(* Schneider Machine Expert - Basic project Ladder Programming_Devin Ezekiel Purba_2106701583, file version 2.7.0.0 *)
(* ProjectInformations: Name=New project *)

HARDWARE
  Cpu 0: TM221C16R
  EthernetConfiguration: NetworkName=M221, IpAllocationMode=FixedAddress, IpAddress=0.0.0.0, SubnetMask=0.0.0.0
  SerialLineConfiguration: Baud=Baud19200, Parity=ParityEven, DataBits=DataBits8, StopBits=StopBits1, PhysicalMedium=PhysicalMediumRs485, TransmissionMode=TransmissionModeModbusRtu, SlaveId=1, Addressing=SlaveAddressing
  MastTask: UsePeriodScanMode=false, PeriodScan=100
  FastTask: Period=255
  CpuBehavior: StartingMode=StartAsPreviousState, AutoSaveRamOnEeprom=true, WatchdogPeriod=250

SYMBOLS  (address, symbol, comment, settings)
  %M0       RUNNING
  %M1       MC_1_BUSY
  %M2       RETRO_1
  %M3       MC_2_BUSY
  %M4       RETRO_2
  %M5       MC_3_BUSY
  %M6       RETRO_5
  %M7       MC_4_BUSY
  %M8       RETRO_6
  %M9       MC_5_BUSY
  %M10      RETRO_9
  %M11      MC_6_BUSY
  %M12      RETRO_10
  %M13      DIFFUSE_1
  %M14      DIFFUSE_3
  %M15      CLAMPED_1
  %M16      DIFFUSE_2
  %M17      DIFFUSE_4
  %M18      CLAMPED_3
  %M19      DIFFUSE_5
  %M20      DIFFUSE_6
  %M21      CLAMPED_5
  %M22      VISION_BLUE
  %M23      VISION_GREEN
  %M24      VISION_METAL
  %M101     MEMORI_1
  %M102     ITEM_GRABBED_3
  %M103     MEMORI_2
  %M104     MEMORI_3
  %M105     MEMORI_4
  %M106     MEMORI_5
  %M107     MEMORI_6
  %M108     MEMORI_7
  %M109     MEMORI_8
  %M110     MEMORI_9
  %M111     MEMORI_10
  %M112     MEMORI_11
  %M113     MEMORI_12
  %M114     MEMORI_13
  %M115     MEMORI_14
  %M116     MEMORI_15
  %M117     MEMORI_METAL
  %M118     MEMORI_GREEN
  %M119     MEMORI_BLUE
  %M200     CONV_2_14
  %M201     MC_START_1
  %M202     CONV_2_13
  %M203     CONV_2_16
  %M204     MC_START_2
  %M205     CONV_2_15
  %M206     CONV_2_6
  %M207     MC_START_3
  %M208     CONV_2_5
  %M209     CONV_2_8
  %M210     MC_START_4
  %M211     CONV_2_7
  %M212     CONV_2_24
  %M213     MC_START_5
  %M214     CONV_2_23
  %M215     CONV_2_26
  %M216     MC_START_6
  %M217     CONV_2_25
  %M218     CONV_2_9
  %M219     GRAB_3
  %M220     RIGHT_POS_1
  %M221     RIGHT_POS_2
  %M222     CONV_2_11
  %M223     MOVE_Z_3
  %M224     MOVE_X_3
  %M225     RAISE_2
  %M226     CONV_2_10
  %M227     CONV_2_1
  %M228     GRAB_1
  %M229     RIGHT_POS_3
  %M230     RIGHT_POS_4
  %M231     CONV_2_3
  %M232     MOVE_Z_1
  %M233     MOVE_X_1
  %M234     RAISE_4
  %M235     CONV_2_2
  %M236     CONV_2_19
  %M237     GRAB_2
  %M238     RIGHT_POS_5
  %M239     RIGHT_POS_6
  %M240     CONV_2_21
  %M241     MOVE_Z_2
  %M242     MOVE_X_2
  %M243     RAISE_6
  %M244     CONV_2_20
  %M251     CONV_4_10
  %M252     CONV_4_11
  %M253     CONV_4_12
  %M254     PIVOT_TURN_1
  %M255     PIVOT_BELT_1
  %M256     PIVOT_TURN_2
  %M257     PIVOT_BELT_2
  %M258     PIVOT_TURN_3
  %M259     PIVOT_BELT_3
  %M300     CONV_4_1
  %M301     CONV_4_2
  %M302     CONV_4_3
  %M303     CONV_4_4
  %M304     CONV_4_5
  %M305     CONV_4_6
  %M306     CONV_4_7
  %M307     CONV_4_8
  %M308     CONV_4_9
  %M309     CONV_6_1
  %M310     CONV_6_2
  %M311     CONV_6_3
  %M312     CONV_6_4
  %M313     CONV_6_5
  %M314     CONV_2_17
  %M315     CONV_2_18
  %M316     CONV_2_27
  %MW0      XSP1
  %MW1      ZSP1
  %MW2      XSP2
  %MW3      ZSP2
  %MW4      XSP3
  %MW5      ZSP3
  %MW64     X_SP_1
  %MW65     Z_SP_1
  %MW66     X_SP_2
  %MW67     Z_SP_2
  %MW68     X_SP_3
  %MW69     Z_SP_3
  %TM0      TIMER_1  [Preset=3, Base=OneSecond]
  %TM1      TIMER_2  [Preset=3, Base=OneSecond]
  %TM2      TIMER_3  [Preset=3, Base=OneSecond]
  %TM3      TIMER_4  [Preset=3, Base=OneSecond]
  %TM4      TIMER_5  [Preset=3, Base=OneSecond]
  %TM5      TIMER_6  [Preset=3, Base=OneSecond]
  %TM6      TIMER_7  [Preset=10, Base=OneSecond]
  %TM7      TIMER_8  [Preset=10, Base=OneSecond]
  %TM8        [Preset=1, Base=OneHundredMilliSeconds]
  %TM9        [Preset=1, Base=OneHundredMilliSeconds]
  %TM10       [Preset=1, Base=OneSecond]
  %TM11       [Preset=1, Base=OneSecond]
  %TM12       [Preset=1, Base=OneSecond]
  %TM13       [Preset=1, Base=OneSecond]
  %TM14       [Preset=1, Base=OneSecond]
  %TM15       [Preset=1, Base=OneSecond]
  %TM16       [Preset=1, Base=OneSecond]
  %TM17       [Preset=1, Base=OneSecond]
  %TM18       [Preset=1, Base=OneSecond]
  %TM19       [Preset=1, Base=OneSecond]
  %TM20       [Preset=1, Base=OneSecond]
  %TM21       [Preset=1, Base=OneSecond]
  %TM22       [Preset=1, Base=OneSecond]
  %TM23       [Preset=1, Base=OneHundredMilliSeconds]
  %TM24       [Preset=10, Base=OneSecond]
  %TM25       [Preset=1, Base=OneSecond]
  %TM26       [Preset=1, Base=OneSecond]
  %TM27       [Preset=1, Base=OneSecond]
  %TM28       [Preset=1, Base=OneSecond]
  %TM29       [Preset=1, Base=OneSecond]
  %TM30       [Preset=1, Base=OneSecond]
  %TM31       [Preset=1, Base=OneSecond]
  %TM32       [Preset=1, Base=OneSecond]
  %TM33       [Preset=1, Base=OneHundredMilliSeconds]
  %TM34       [Preset=10, Base=OneSecond]
  %TM35       [Preset=1, Base=OneHundredMilliSeconds]
  %TM36       [Preset=10, Base=OneSecond]
  %TM37       [Preset=1, Base=OneSecond]
  %TM38       [Preset=1, Base=OneSecond]
  %TM39       [Preset=1, Base=OneSecond]
  %TM40       [Preset=1, Base=OneSecond]
  %TM41       [Preset=1, Base=OneSecond]
  %TM42       [Preset=1, Base=OneSecond]
  %TM43       [Preset=1, Base=OneSecond]
  %TM44       [Preset=1, Base=OneSecond]
  %TM45       [Preset=1, Base=OneHundredMilliSeconds]
  %TM46       [Preset=10, Base=OneSecond]
  %TM47       [Preset=20, Base=OneHundredMilliSeconds]
  %TM48       [Preset=1, Base=OneSecond]
  %TM49       [Preset=2, Base=OneSecond]

POU Production
  (* SectionNumber=1 *)

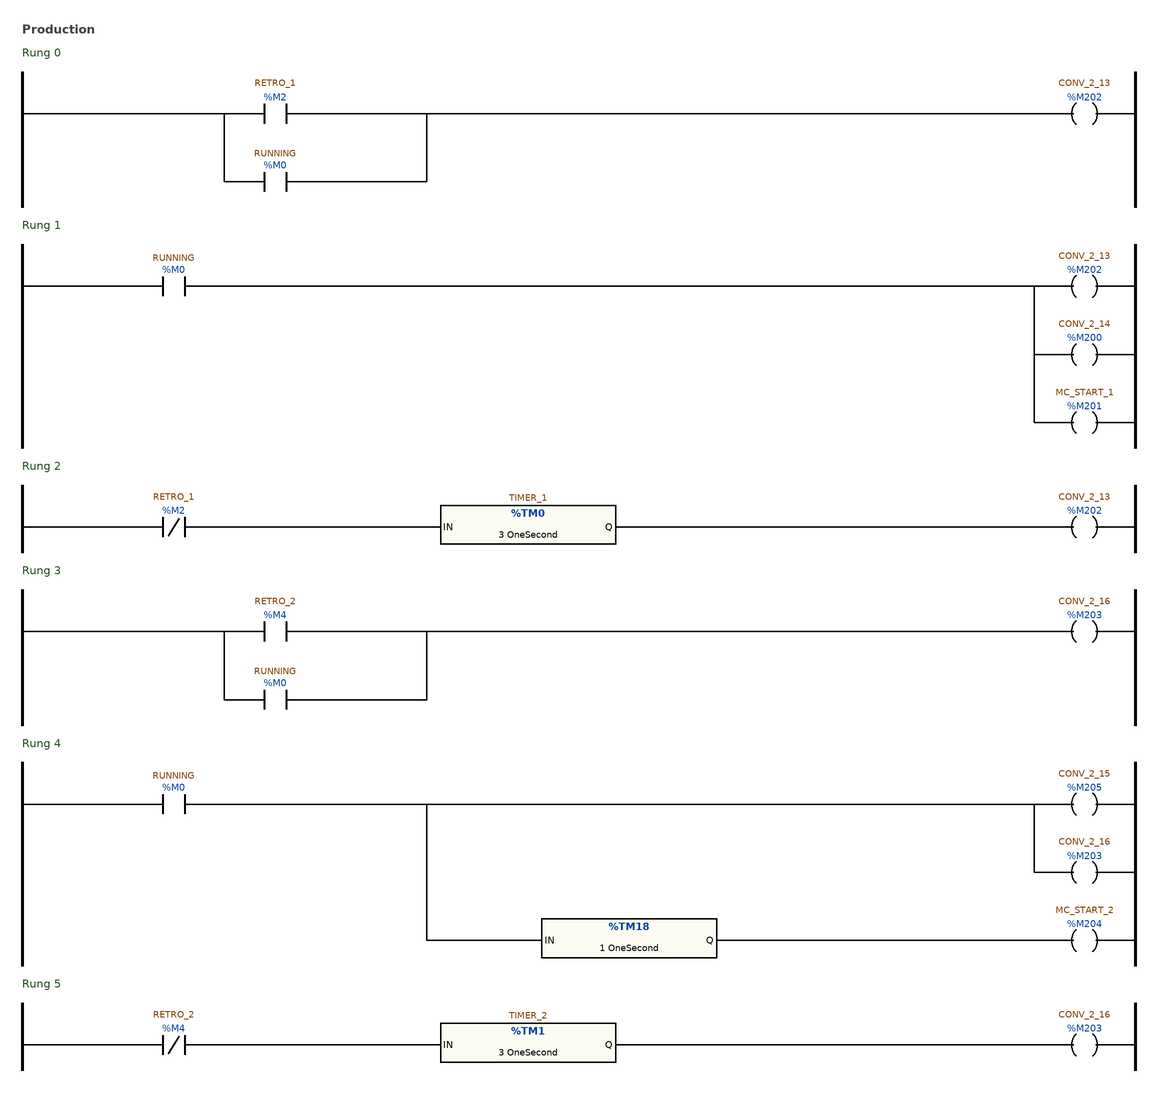

// Rung 0
  LD 1
  AND( %M2                (* RETRO_1 *)
  OR %M0                  (* RUNNING *)
  )
  ST %M202                (* CONV_2_13 *)
  // as ST:
  //   CONV_2_13 := RETRO_1 OR RUNNING;

// Rung 1
  LD %M0                  (* RUNNING *)
  ST %M202                (* CONV_2_13 *)
  ST %M200                (* CONV_2_14 *)
  ST %M201                (* MC_START_1 *)
  // as ST:
  //   CONV_2_13 := RUNNING;
  //   CONV_2_14 := RUNNING;
  //   MC_START_1 := RUNNING;

// Rung 2
  BLK %TM0                (* TIMER_1 *)
  LDN %M2                 (* RETRO_1 *)
  IN
  OUT_BLK
  LD Q
  ST %M202                (* CONV_2_13 *)
  END_BLK
  // as ST:
  //   TIMER_1(IN := NOT RETRO_1);
  //   CONV_2_13 := TIMER_1.Q;

// Rung 3
  LD 1
  AND( %M4                (* RETRO_2 *)
  OR %M0                  (* RUNNING *)
  )
  ST %M203                (* CONV_2_16 *)
  // as ST:
  //   CONV_2_16 := RETRO_2 OR RUNNING;

// Rung 4
  LD 1
  MULTIFB
  LD 1
  AND %M0                 (* RUNNING *)
  ST %MW2009:X0
  LD %MW2009:X0
  ST %M205                (* CONV_2_15 *)
  ST %M203                (* CONV_2_16 *)
  BLK %TM18
  LD %MW2009:X0
  IN
  OUT_BLK
  LD Q
  ST %M204                (* MC_START_2 *)
  END_BLK
  MULTIFB
  // as ST:
  //   CONV_2_15 := RUNNING;
  //   CONV_2_16 := RUNNING;
  //   %TM18(IN := RUNNING);
  //   MC_START_2 := %TM18.Q;

// Rung 5
  BLK %TM1                (* TIMER_2 *)
  LDN %M4                 (* RETRO_2 *)
  IN
  OUT_BLK
  LD Q
  ST %M203                (* CONV_2_16 *)
  END_BLK
  // as ST:
  //   TIMER_2(IN := NOT RETRO_2);
  //   CONV_2_16 := TIMER_2.Q;

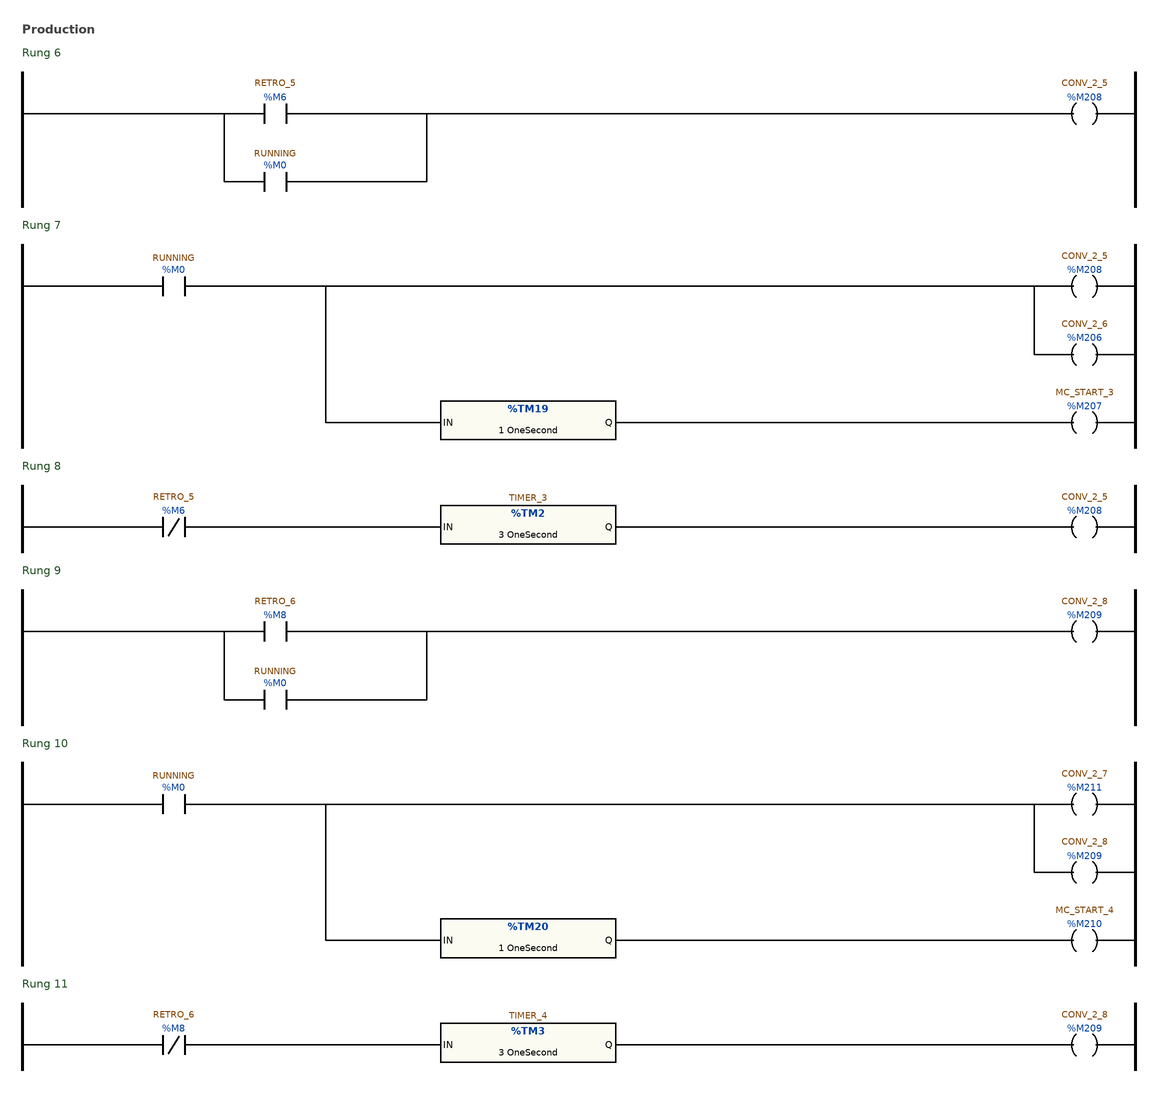

// Rung 6
  LD 1
  AND( %M6                (* RETRO_5 *)
  OR %M0                  (* RUNNING *)
  )
  ST %M208                (* CONV_2_5 *)
  // as ST:
  //   CONV_2_5 := RETRO_5 OR RUNNING;

// Rung 7
  LD 1
  MULTIFB
  LD 1
  AND %M0                 (* RUNNING *)
  ST %MW2009:X0
  LD %MW2009:X0
  ST %M208                (* CONV_2_5 *)
  ST %M206                (* CONV_2_6 *)
  BLK %TM19
  LD %MW2009:X0
  IN
  OUT_BLK
  LD Q
  ST %M207                (* MC_START_3 *)
  END_BLK
  MULTIFB
  // as ST:
  //   CONV_2_5 := RUNNING;
  //   CONV_2_6 := RUNNING;
  //   %TM19(IN := RUNNING);
  //   MC_START_3 := %TM19.Q;

// Rung 8
  BLK %TM2                (* TIMER_3 *)
  LDN %M6                 (* RETRO_5 *)
  IN
  OUT_BLK
  LD Q
  ST %M208                (* CONV_2_5 *)
  END_BLK
  // as ST:
  //   TIMER_3(IN := NOT RETRO_5);
  //   CONV_2_5 := TIMER_3.Q;

// Rung 9
  LD 1
  AND( %M8                (* RETRO_6 *)
  OR %M0                  (* RUNNING *)
  )
  ST %M209                (* CONV_2_8 *)
  // as ST:
  //   CONV_2_8 := RETRO_6 OR RUNNING;

// Rung 10
  LD 1
  MULTIFB
  LD 1
  AND %M0                 (* RUNNING *)
  ST %MW2009:X0
  LD %MW2009:X0
  ST %M211                (* CONV_2_7 *)
  ST %M209                (* CONV_2_8 *)
  BLK %TM20
  LD %MW2009:X0
  IN
  OUT_BLK
  LD Q
  ST %M210                (* MC_START_4 *)
  END_BLK
  MULTIFB
  // as ST:
  //   CONV_2_7 := RUNNING;
  //   CONV_2_8 := RUNNING;
  //   %TM20(IN := RUNNING);
  //   MC_START_4 := %TM20.Q;

// Rung 11
  BLK %TM3                (* TIMER_4 *)
  LDN %M8                 (* RETRO_6 *)
  IN
  OUT_BLK
  LD Q
  ST %M209                (* CONV_2_8 *)
  END_BLK
  // as ST:
  //   TIMER_4(IN := NOT RETRO_6);
  //   CONV_2_8 := TIMER_4.Q;

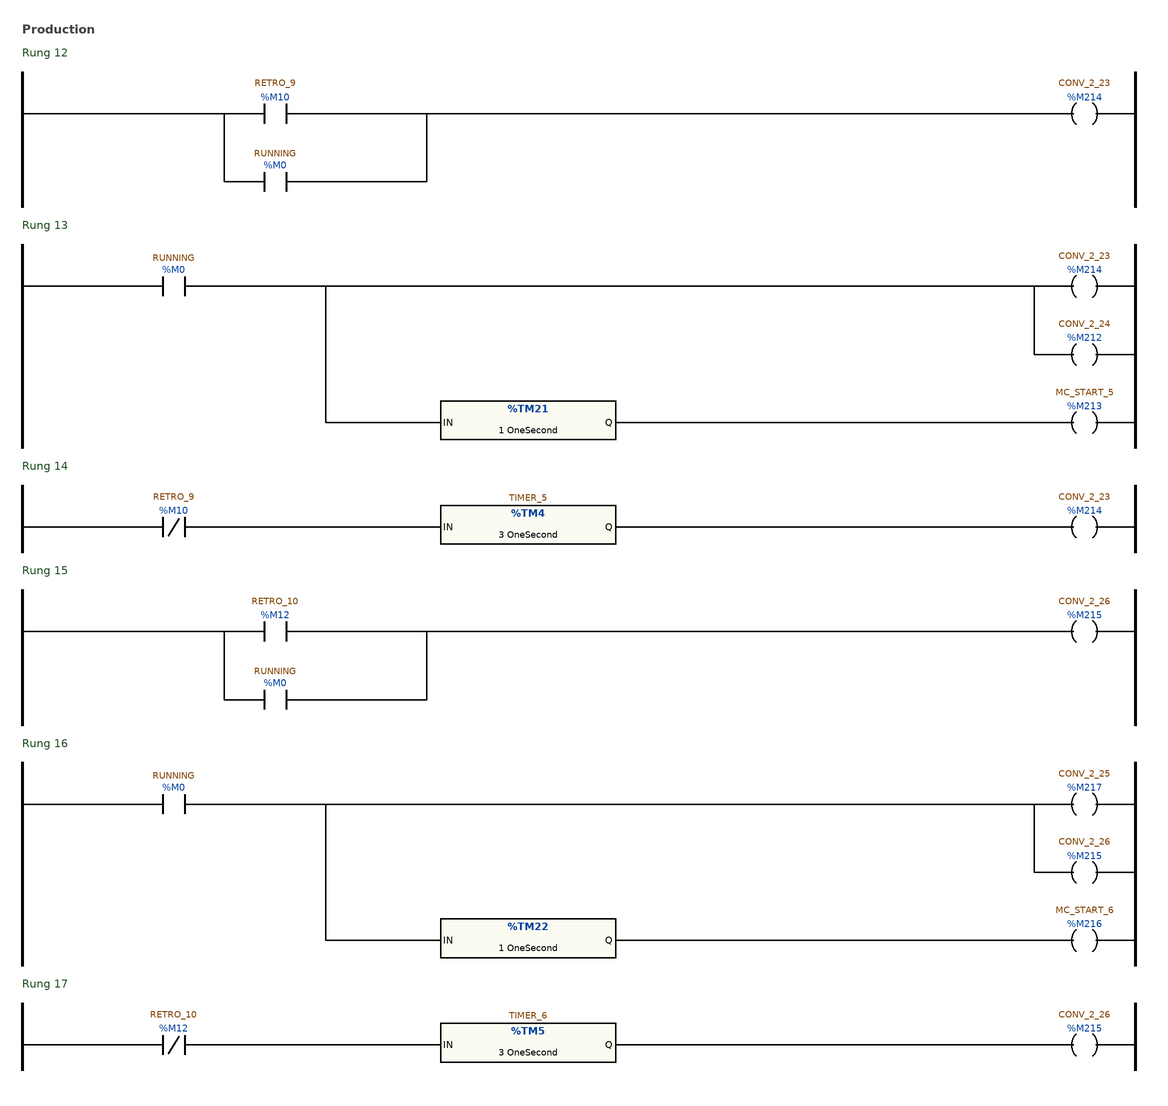

// Rung 12
  LD 1
  AND( %M10               (* RETRO_9 *)
  OR %M0                  (* RUNNING *)
  )
  ST %M214                (* CONV_2_23 *)
  // as ST:
  //   CONV_2_23 := RETRO_9 OR RUNNING;

// Rung 13
  LD 1
  MULTIFB
  LD 1
  AND %M0                 (* RUNNING *)
  ST %MW2009:X0
  LD %MW2009:X0
  ST %M214                (* CONV_2_23 *)
  ST %M212                (* CONV_2_24 *)
  BLK %TM21
  LD %MW2009:X0
  IN
  OUT_BLK
  LD Q
  ST %M213                (* MC_START_5 *)
  END_BLK
  MULTIFB
  // as ST:
  //   CONV_2_23 := RUNNING;
  //   CONV_2_24 := RUNNING;
  //   %TM21(IN := RUNNING);
  //   MC_START_5 := %TM21.Q;

// Rung 14
  BLK %TM4                (* TIMER_5 *)
  LDN %M10                (* RETRO_9 *)
  IN
  OUT_BLK
  LD Q
  ST %M214                (* CONV_2_23 *)
  END_BLK
  // as ST:
  //   TIMER_5(IN := NOT RETRO_9);
  //   CONV_2_23 := TIMER_5.Q;

// Rung 15
  LD 1
  AND( %M12               (* RETRO_10 *)
  OR %M0                  (* RUNNING *)
  )
  ST %M215                (* CONV_2_26 *)
  // as ST:
  //   CONV_2_26 := RETRO_10 OR RUNNING;

// Rung 16
  LD 1
  MULTIFB
  LD 1
  AND %M0                 (* RUNNING *)
  ST %MW2009:X0
  LD %MW2009:X0
  ST %M217                (* CONV_2_25 *)
  ST %M215                (* CONV_2_26 *)
  BLK %TM22
  LD %MW2009:X0
  IN
  OUT_BLK
  LD Q
  ST %M216                (* MC_START_6 *)
  END_BLK
  MULTIFB
  // as ST:
  //   CONV_2_25 := RUNNING;
  //   CONV_2_26 := RUNNING;
  //   %TM22(IN := RUNNING);
  //   MC_START_6 := %TM22.Q;

// Rung 17
  BLK %TM5                (* TIMER_6 *)
  LDN %M12                (* RETRO_10 *)
  IN
  OUT_BLK
  LD Q
  ST %M215                (* CONV_2_26 *)
  END_BLK
  // as ST:
  //   TIMER_6(IN := NOT RETRO_10);
  //   CONV_2_26 := TIMER_6.Q;

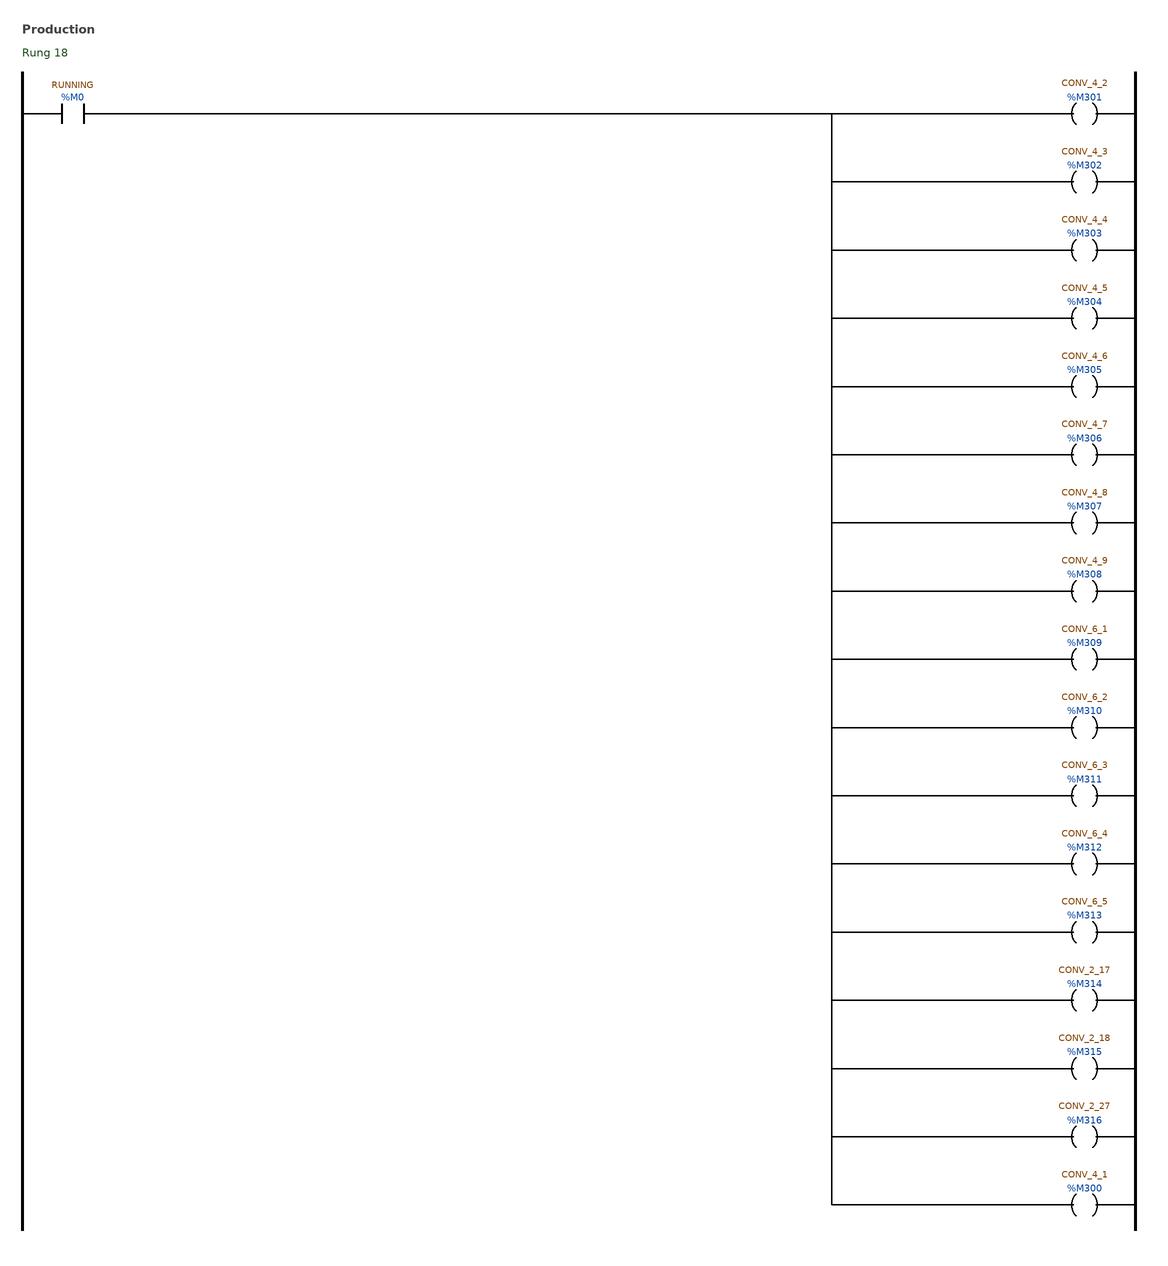

// Rung 18
  LD %M0                  (* RUNNING *)
  ST %M301                (* CONV_4_2 *)
  ST %M302                (* CONV_4_3 *)
  ST %M303                (* CONV_4_4 *)
  ST %M304                (* CONV_4_5 *)
  ST %M305                (* CONV_4_6 *)
  ST %M306                (* CONV_4_7 *)
  ST %M307                (* CONV_4_8 *)
  ST %M308                (* CONV_4_9 *)
  ST %M309                (* CONV_6_1 *)
  ST %M310                (* CONV_6_2 *)
  ST %M311                (* CONV_6_3 *)
  ST %M312                (* CONV_6_4 *)
  ST %M313                (* CONV_6_5 *)
  ST %M314                (* CONV_2_17 *)
  ST %M315                (* CONV_2_18 *)
  ST %M316                (* CONV_2_27 *)
  ST %M300                (* CONV_4_1 *)
  // as ST:
  //   CONV_4_2 := RUNNING;
  //   CONV_4_3 := RUNNING;
  //   CONV_4_4 := RUNNING;
  //   CONV_4_5 := RUNNING;
  //   CONV_4_6 := RUNNING;
  //   CONV_4_7 := RUNNING;
  //   CONV_4_8 := RUNNING;
  //   CONV_4_9 := RUNNING;
  //   CONV_6_1 := RUNNING;
  //   CONV_6_2 := RUNNING;
  //   CONV_6_3 := RUNNING;
  //   CONV_6_4 := RUNNING;
  //   CONV_6_5 := RUNNING;
  //   CONV_2_17 := RUNNING;
  //   CONV_2_18 := RUNNING;
  //   CONV_2_27 := RUNNING;
  //   CONV_4_1 := RUNNING;

POU Assembler
  (* SectionNumber=2 *)

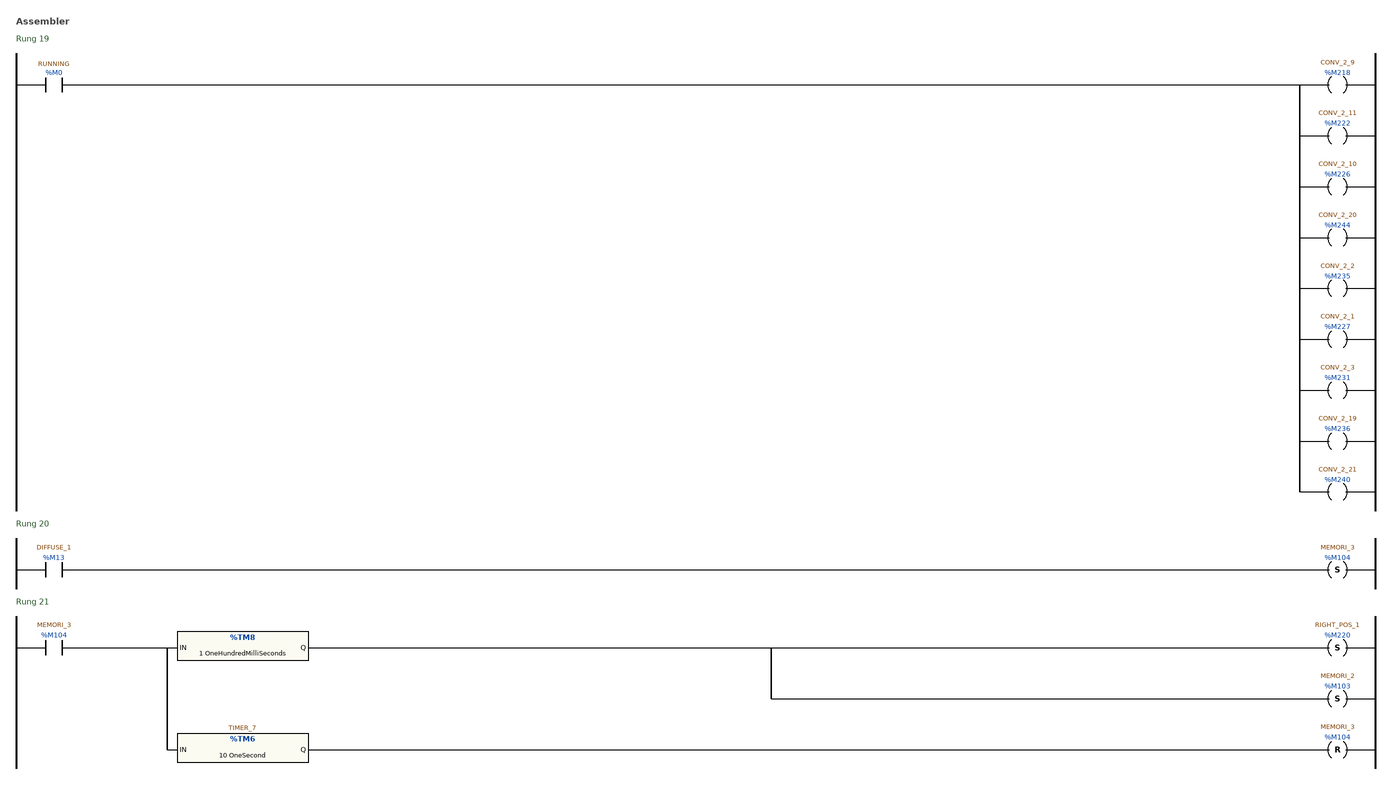

// Rung 19
  LD %M0                  (* RUNNING *)
  ST %M218                (* CONV_2_9 *)
  ST %M222                (* CONV_2_11 *)
  ST %M226                (* CONV_2_10 *)
  ST %M244                (* CONV_2_20 *)
  ST %M235                (* CONV_2_2 *)
  ST %M227                (* CONV_2_1 *)
  ST %M231                (* CONV_2_3 *)
  ST %M236                (* CONV_2_19 *)
  ST %M240                (* CONV_2_21 *)
  // as ST:
  //   CONV_2_9 := RUNNING;
  //   CONV_2_11 := RUNNING;
  //   CONV_2_10 := RUNNING;
  //   CONV_2_20 := RUNNING;
  //   CONV_2_2 := RUNNING;
  //   CONV_2_1 := RUNNING;
  //   CONV_2_3 := RUNNING;
  //   CONV_2_19 := RUNNING;
  //   CONV_2_21 := RUNNING;

// Rung 20
  LD %M13                 (* DIFFUSE_1 *)
  S %M104                 (* MEMORI_3 *)
  // as ST:
  //   IF DIFFUSE_1 THEN MEMORI_3 := TRUE; END_IF;

// Rung 21
  LD 1
  MULTIFB
  LD 1
  AND %M104               (* MEMORI_3 *)
  ST %MW2009:X0
  BLK %TM8
  LD %MW2009:X0
  IN
  OUT_BLK
  LD Q
  S %M220                 (* RIGHT_POS_1 *)
  S %M103                 (* MEMORI_2 *)
  END_BLK
  BLK %TM6                (* TIMER_7 *)
  LD %MW2009:X0
  IN
  OUT_BLK
  LD Q
  R %M104                 (* MEMORI_3 *)
  END_BLK
  MULTIFB
  // as ST:
  //   %TM8(IN := MEMORI_3);
  //   IF %TM8.Q THEN RIGHT_POS_1 := TRUE; END_IF;
  //   IF %TM8.Q THEN MEMORI_2 := TRUE; END_IF;
  //   TIMER_7(IN := MEMORI_3);
  //   IF TIMER_7.Q THEN MEMORI_3 := FALSE; END_IF;

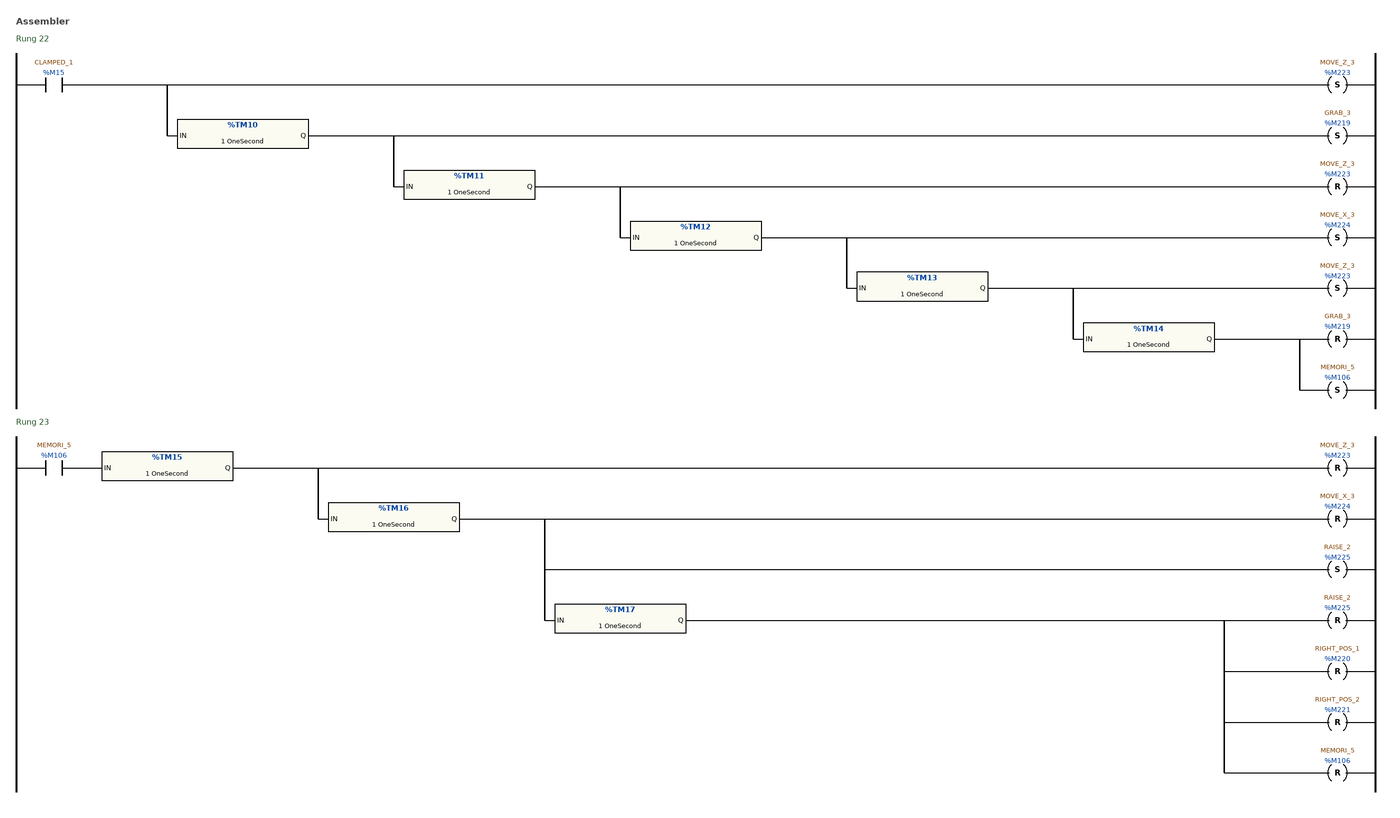

// Rung 22
  LD 1
  MULTIFB
  LD 1
  AND %M15                (* CLAMPED_1 *)
  ST %MW2009:X4
  LD %MW2009:X4
  S %M223                 (* MOVE_Z_3 *)
  BLK %TM10
  LD %MW2009:X4
  IN
  OUT_BLK
  LD Q
  ST %MW2009:X0
  END_BLK
  LD %MW2009:X0
  S %M219                 (* GRAB_3 *)
  BLK %TM11
  LD %MW2009:X0
  IN
  OUT_BLK
  LD Q
  ST %MW2009:X1
  END_BLK
  LD %MW2009:X1
  R %M223                 (* MOVE_Z_3 *)
  BLK %TM12
  LD %MW2009:X1
  IN
  OUT_BLK
  LD Q
  ST %MW2009:X2
  END_BLK
  LD %MW2009:X2
  S %M224                 (* MOVE_X_3 *)
  BLK %TM13
  LD %MW2009:X2
  IN
  OUT_BLK
  LD Q
  ST %MW2009:X3
  END_BLK
  LD %MW2009:X3
  S %M223                 (* MOVE_Z_3 *)
  BLK %TM14
  LD %MW2009:X3
  IN
  OUT_BLK
  LD Q
  R %M219                 (* GRAB_3 *)
  S %M106                 (* MEMORI_5 *)
  END_BLK
  MULTIFB
  // as ST:
  //   IF CLAMPED_1 THEN MOVE_Z_3 := TRUE; END_IF;
  //   %TM10(IN := CLAMPED_1);
  //   IF %TM10.Q THEN GRAB_3 := TRUE; END_IF;
  //   %TM11(IN := %TM10.Q);
  //   IF %TM11.Q THEN MOVE_Z_3 := FALSE; END_IF;
  //   %TM12(IN := %TM11.Q);
  //   IF %TM12.Q THEN MOVE_X_3 := TRUE; END_IF;
  //   %TM13(IN := %TM12.Q);
  //   IF %TM13.Q THEN MOVE_Z_3 := TRUE; END_IF;
  //   %TM14(IN := %TM13.Q);
  //   IF %TM14.Q THEN GRAB_3 := FALSE; END_IF;
  //   IF %TM14.Q THEN MEMORI_5 := TRUE; END_IF;

// Rung 23
  LD 1
  MULTIFB
  BLK %TM15
  LD 1
  AND %M106               (* MEMORI_5 *)
  IN
  OUT_BLK
  LD Q
  ST %MW2009:X0
  END_BLK
  LD %MW2009:X0
  R %M223                 (* MOVE_Z_3 *)
  BLK %TM16
  LD %MW2009:X0
  IN
  OUT_BLK
  LD Q
  ST %MW2009:X1
  END_BLK
  LD %MW2009:X1
  R %M224                 (* MOVE_X_3 *)
  S %M225                 (* RAISE_2 *)
  BLK %TM17
  LD %MW2009:X1
  IN
  OUT_BLK
  LD Q
  R %M225                 (* RAISE_2 *)
  R %M220                 (* RIGHT_POS_1 *)
  R %M221                 (* RIGHT_POS_2 *)
  R %M106                 (* MEMORI_5 *)
  END_BLK
  MULTIFB
  // as ST:
  //   %TM15(IN := MEMORI_5);
  //   IF %TM15.Q THEN MOVE_Z_3 := FALSE; END_IF;
  //   %TM16(IN := %TM15.Q);
  //   IF %TM16.Q THEN MOVE_X_3 := FALSE; END_IF;
  //   IF %TM16.Q THEN RAISE_2 := TRUE; END_IF;
  //   %TM17(IN := %TM16.Q);
  //   IF %TM17.Q THEN RAISE_2 := FALSE; END_IF;
  //   IF %TM17.Q THEN RIGHT_POS_1 := FALSE; END_IF;
  //   IF %TM17.Q THEN RIGHT_POS_2 := FALSE; END_IF;
  //   IF %TM17.Q THEN MEMORI_5 := FALSE; END_IF;

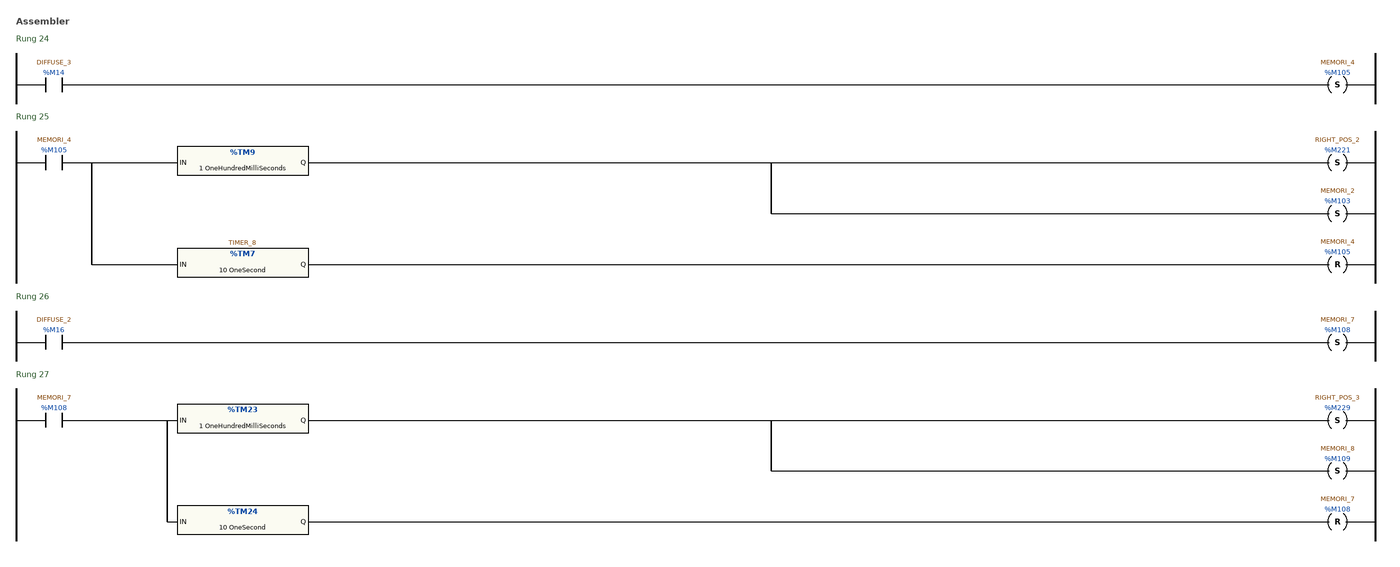

// Rung 24
  LD %M14                 (* DIFFUSE_3 *)
  S %M105                 (* MEMORI_4 *)
  // as ST:
  //   IF DIFFUSE_3 THEN MEMORI_4 := TRUE; END_IF;

// Rung 25
  LD 1
  MULTIFB
  LD 1
  AND %M105               (* MEMORI_4 *)
  ST %MW2009:X0
  BLK %TM9
  LD %MW2009:X0
  IN
  OUT_BLK
  LD Q
  S %M221                 (* RIGHT_POS_2 *)
  S %M103                 (* MEMORI_2 *)
  END_BLK
  BLK %TM7                (* TIMER_8 *)
  LD %MW2009:X0
  IN
  OUT_BLK
  LD Q
  R %M105                 (* MEMORI_4 *)
  END_BLK
  MULTIFB
  // as ST:
  //   %TM9(IN := MEMORI_4);
  //   IF %TM9.Q THEN RIGHT_POS_2 := TRUE; END_IF;
  //   IF %TM9.Q THEN MEMORI_2 := TRUE; END_IF;
  //   TIMER_8(IN := MEMORI_4);
  //   IF TIMER_8.Q THEN MEMORI_4 := FALSE; END_IF;

// Rung 26
  LD %M16                 (* DIFFUSE_2 *)
  S %M108                 (* MEMORI_7 *)
  // as ST:
  //   IF DIFFUSE_2 THEN MEMORI_7 := TRUE; END_IF;

// Rung 27
  LD 1
  MULTIFB
  LD 1
  AND %M108               (* MEMORI_7 *)
  ST %MW2009:X0
  BLK %TM23
  LD %MW2009:X0
  IN
  OUT_BLK
  LD Q
  S %M229                 (* RIGHT_POS_3 *)
  S %M109                 (* MEMORI_8 *)
  END_BLK
  BLK %TM24
  LD %MW2009:X0
  IN
  OUT_BLK
  LD Q
  R %M108                 (* MEMORI_7 *)
  END_BLK
  MULTIFB
  // as ST:
  //   %TM23(IN := MEMORI_7);
  //   IF %TM23.Q THEN RIGHT_POS_3 := TRUE; END_IF;
  //   IF %TM23.Q THEN MEMORI_8 := TRUE; END_IF;
  //   %TM24(IN := MEMORI_7);
  //   IF %TM24.Q THEN MEMORI_7 := FALSE; END_IF;

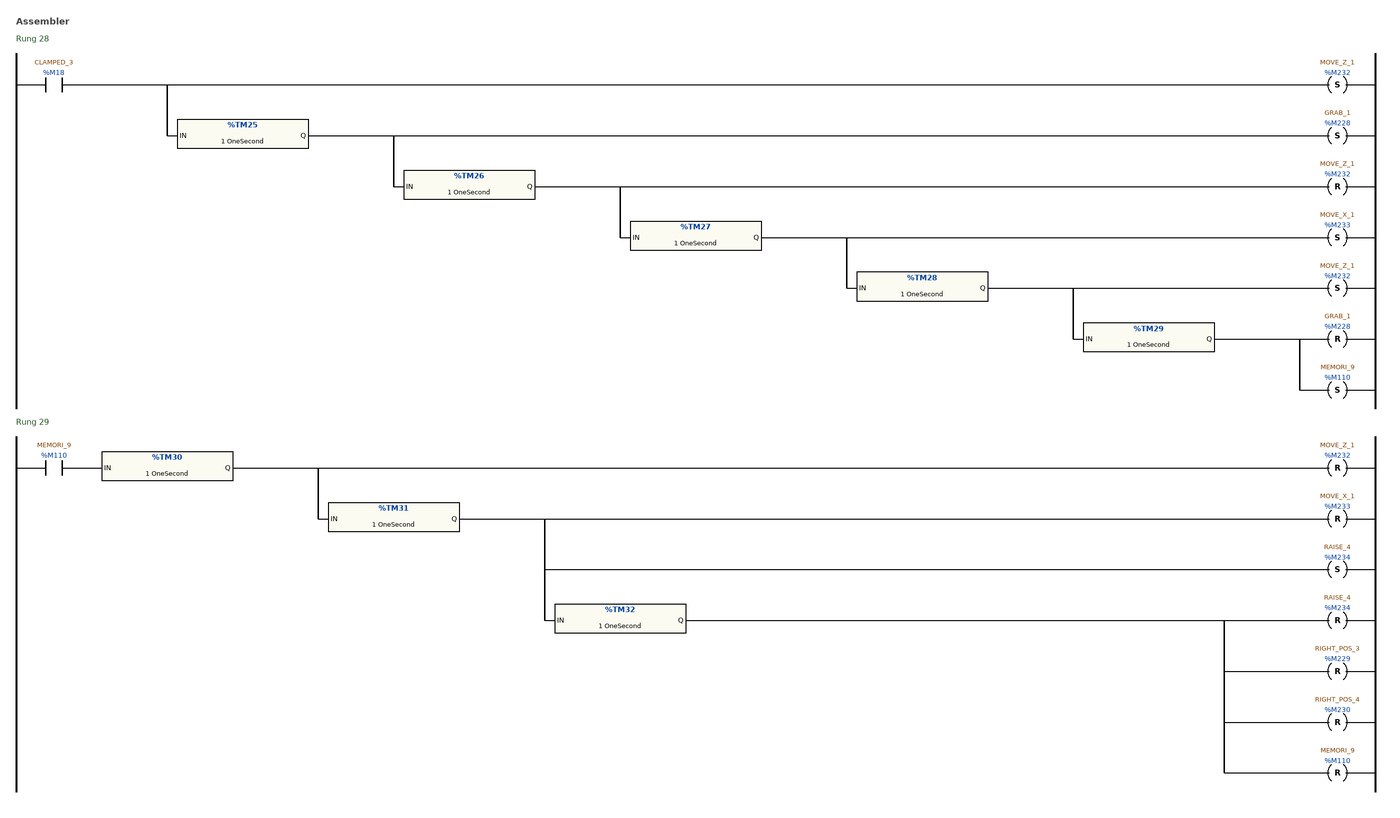

// Rung 28
  LD 1
  MULTIFB
  LD 1
  AND %M18                (* CLAMPED_3 *)
  ST %MW2009:X4
  LD %MW2009:X4
  S %M232                 (* MOVE_Z_1 *)
  BLK %TM25
  LD %MW2009:X4
  IN
  OUT_BLK
  LD Q
  ST %MW2009:X0
  END_BLK
  LD %MW2009:X0
  S %M228                 (* GRAB_1 *)
  BLK %TM26
  LD %MW2009:X0
  IN
  OUT_BLK
  LD Q
  ST %MW2009:X1
  END_BLK
  LD %MW2009:X1
  R %M232                 (* MOVE_Z_1 *)
  BLK %TM27
  LD %MW2009:X1
  IN
  OUT_BLK
  LD Q
  ST %MW2009:X2
  END_BLK
  LD %MW2009:X2
  S %M233                 (* MOVE_X_1 *)
  BLK %TM28
  LD %MW2009:X2
  IN
  OUT_BLK
  LD Q
  ST %MW2009:X3
  END_BLK
  LD %MW2009:X3
  S %M232                 (* MOVE_Z_1 *)
  BLK %TM29
  LD %MW2009:X3
  IN
  OUT_BLK
  LD Q
  R %M228                 (* GRAB_1 *)
  S %M110                 (* MEMORI_9 *)
  END_BLK
  MULTIFB
  // as ST:
  //   IF CLAMPED_3 THEN MOVE_Z_1 := TRUE; END_IF;
  //   %TM25(IN := CLAMPED_3);
  //   IF %TM25.Q THEN GRAB_1 := TRUE; END_IF;
  //   %TM26(IN := %TM25.Q);
  //   IF %TM26.Q THEN MOVE_Z_1 := FALSE; END_IF;
  //   %TM27(IN := %TM26.Q);
  //   IF %TM27.Q THEN MOVE_X_1 := TRUE; END_IF;
  //   %TM28(IN := %TM27.Q);
  //   IF %TM28.Q THEN MOVE_Z_1 := TRUE; END_IF;
  //   %TM29(IN := %TM28.Q);
  //   IF %TM29.Q THEN GRAB_1 := FALSE; END_IF;
  //   IF %TM29.Q THEN MEMORI_9 := TRUE; END_IF;

// Rung 29
  LD 1
  MULTIFB
  BLK %TM30
  LD 1
  AND %M110               (* MEMORI_9 *)
  IN
  OUT_BLK
  LD Q
  ST %MW2009:X0
  END_BLK
  LD %MW2009:X0
  R %M232                 (* MOVE_Z_1 *)
  BLK %TM31
  LD %MW2009:X0
  IN
  OUT_BLK
  LD Q
  ST %MW2009:X1
  END_BLK
  LD %MW2009:X1
  R %M233                 (* MOVE_X_1 *)
  S %M234                 (* RAISE_4 *)
  BLK %TM32
  LD %MW2009:X1
  IN
  OUT_BLK
  LD Q
  R %M234                 (* RAISE_4 *)
  R %M229                 (* RIGHT_POS_3 *)
  R %M230                 (* RIGHT_POS_4 *)
  R %M110                 (* MEMORI_9 *)
  END_BLK
  MULTIFB
  // as ST:
  //   %TM30(IN := MEMORI_9);
  //   IF %TM30.Q THEN MOVE_Z_1 := FALSE; END_IF;
  //   %TM31(IN := %TM30.Q);
  //   IF %TM31.Q THEN MOVE_X_1 := FALSE; END_IF;
  //   IF %TM31.Q THEN RAISE_4 := TRUE; END_IF;
  //   %TM32(IN := %TM31.Q);
  //   IF %TM32.Q THEN RAISE_4 := FALSE; END_IF;
  //   IF %TM32.Q THEN RIGHT_POS_3 := FALSE; END_IF;
  //   IF %TM32.Q THEN RIGHT_POS_4 := FALSE; END_IF;
  //   IF %TM32.Q THEN MEMORI_9 := FALSE; END_IF;

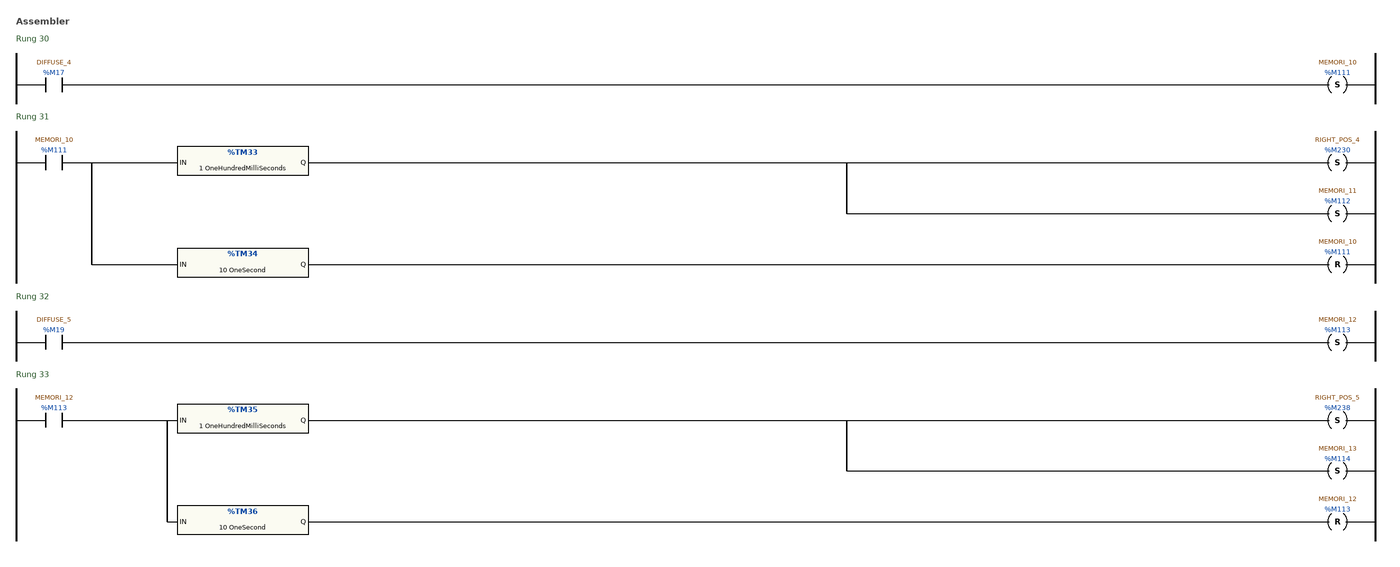

// Rung 30
  LD %M17                 (* DIFFUSE_4 *)
  S %M111                 (* MEMORI_10 *)
  // as ST:
  //   IF DIFFUSE_4 THEN MEMORI_10 := TRUE; END_IF;

// Rung 31
  LD 1
  MULTIFB
  LD 1
  AND %M111               (* MEMORI_10 *)
  ST %MW2009:X0
  BLK %TM33
  LD %MW2009:X0
  IN
  OUT_BLK
  LD Q
  S %M230                 (* RIGHT_POS_4 *)
  S %M112                 (* MEMORI_11 *)
  END_BLK
  BLK %TM34
  LD %MW2009:X0
  IN
  OUT_BLK
  LD Q
  R %M111                 (* MEMORI_10 *)
  END_BLK
  MULTIFB
  // as ST:
  //   %TM33(IN := MEMORI_10);
  //   IF %TM33.Q THEN RIGHT_POS_4 := TRUE; END_IF;
  //   IF %TM33.Q THEN MEMORI_11 := TRUE; END_IF;
  //   %TM34(IN := MEMORI_10);
  //   IF %TM34.Q THEN MEMORI_10 := FALSE; END_IF;

// Rung 32
  LD %M19                 (* DIFFUSE_5 *)
  S %M113                 (* MEMORI_12 *)
  // as ST:
  //   IF DIFFUSE_5 THEN MEMORI_12 := TRUE; END_IF;

// Rung 33
  LD 1
  MULTIFB
  LD 1
  AND %M113               (* MEMORI_12 *)
  ST %MW2009:X0
  BLK %TM35
  LD %MW2009:X0
  IN
  OUT_BLK
  LD Q
  S %M238                 (* RIGHT_POS_5 *)
  S %M114                 (* MEMORI_13 *)
  END_BLK
  BLK %TM36
  LD %MW2009:X0
  IN
  OUT_BLK
  LD Q
  R %M113                 (* MEMORI_12 *)
  END_BLK
  MULTIFB
  // as ST:
  //   %TM35(IN := MEMORI_12);
  //   IF %TM35.Q THEN RIGHT_POS_5 := TRUE; END_IF;
  //   IF %TM35.Q THEN MEMORI_13 := TRUE; END_IF;
  //   %TM36(IN := MEMORI_12);
  //   IF %TM36.Q THEN MEMORI_12 := FALSE; END_IF;

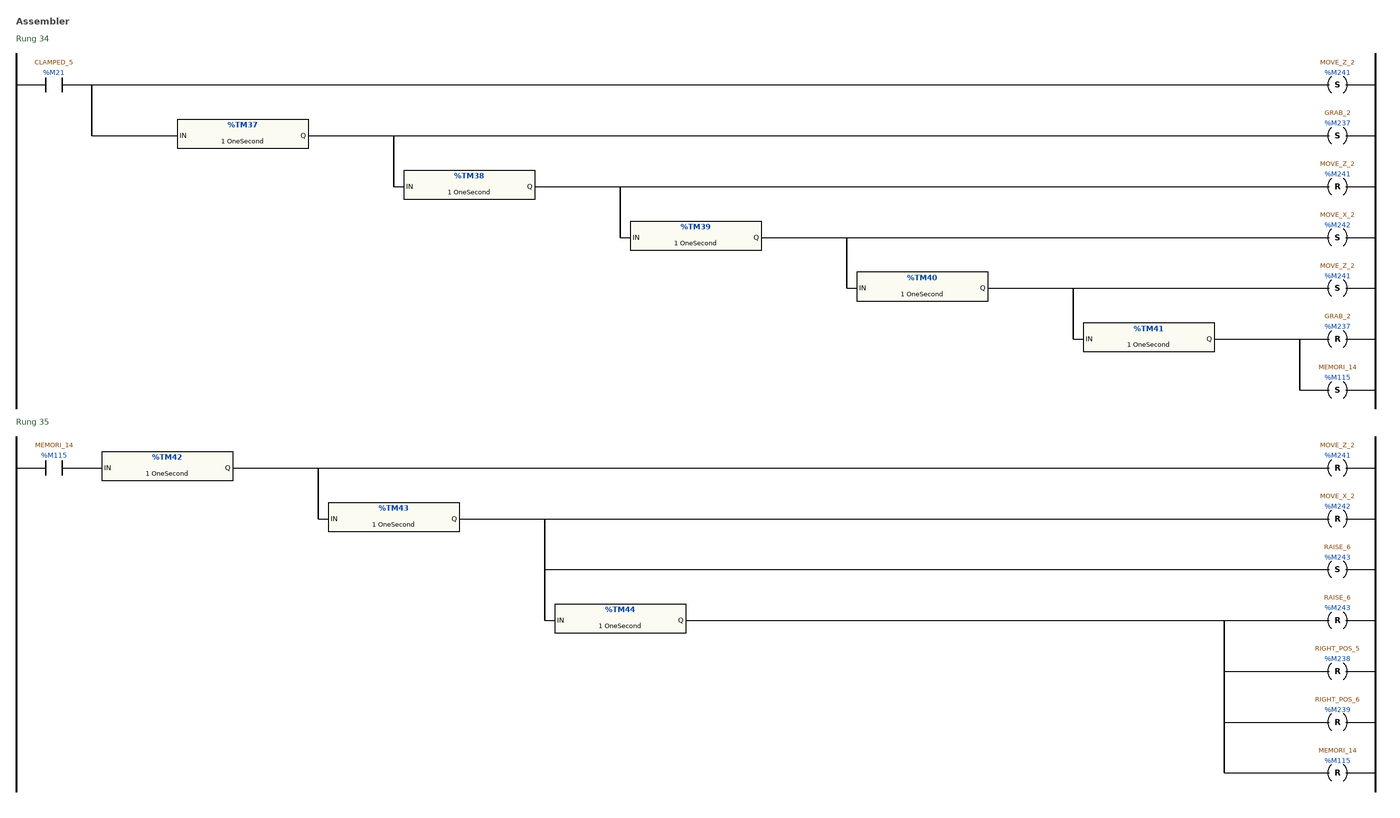

// Rung 34
  LD 1
  MULTIFB
  LD 1
  AND %M21                (* CLAMPED_5 *)
  ST %MW2009:X4
  LD %MW2009:X4
  S %M241                 (* MOVE_Z_2 *)
  BLK %TM37
  LD %MW2009:X4
  IN
  OUT_BLK
  LD Q
  ST %MW2009:X0
  END_BLK
  LD %MW2009:X0
  S %M237                 (* GRAB_2 *)
  BLK %TM38
  LD %MW2009:X0
  IN
  OUT_BLK
  LD Q
  ST %MW2009:X1
  END_BLK
  LD %MW2009:X1
  R %M241                 (* MOVE_Z_2 *)
  BLK %TM39
  LD %MW2009:X1
  IN
  OUT_BLK
  LD Q
  ST %MW2009:X2
  END_BLK
  LD %MW2009:X2
  S %M242                 (* MOVE_X_2 *)
  BLK %TM40
  LD %MW2009:X2
  IN
  OUT_BLK
  LD Q
  ST %MW2009:X3
  END_BLK
  LD %MW2009:X3
  S %M241                 (* MOVE_Z_2 *)
  BLK %TM41
  LD %MW2009:X3
  IN
  OUT_BLK
  LD Q
  R %M237                 (* GRAB_2 *)
  S %M115                 (* MEMORI_14 *)
  END_BLK
  MULTIFB
  // as ST:
  //   IF CLAMPED_5 THEN MOVE_Z_2 := TRUE; END_IF;
  //   %TM37(IN := CLAMPED_5);
  //   IF %TM37.Q THEN GRAB_2 := TRUE; END_IF;
  //   %TM38(IN := %TM37.Q);
  //   IF %TM38.Q THEN MOVE_Z_2 := FALSE; END_IF;
  //   %TM39(IN := %TM38.Q);
  //   IF %TM39.Q THEN MOVE_X_2 := TRUE; END_IF;
  //   %TM40(IN := %TM39.Q);
  //   IF %TM40.Q THEN MOVE_Z_2 := TRUE; END_IF;
  //   %TM41(IN := %TM40.Q);
  //   IF %TM41.Q THEN GRAB_2 := FALSE; END_IF;
  //   IF %TM41.Q THEN MEMORI_14 := TRUE; END_IF;

// Rung 35
  LD 1
  MULTIFB
  BLK %TM42
  LD 1
  AND %M115               (* MEMORI_14 *)
  IN
  OUT_BLK
  LD Q
  ST %MW2009:X0
  END_BLK
  LD %MW2009:X0
  R %M241                 (* MOVE_Z_2 *)
  BLK %TM43
  LD %MW2009:X0
  IN
  OUT_BLK
  LD Q
  ST %MW2009:X1
  END_BLK
  LD %MW2009:X1
  R %M242                 (* MOVE_X_2 *)
  S %M243                 (* RAISE_6 *)
  BLK %TM44
  LD %MW2009:X1
  IN
  OUT_BLK
  LD Q
  R %M243                 (* RAISE_6 *)
  R %M238                 (* RIGHT_POS_5 *)
  R %M239                 (* RIGHT_POS_6 *)
  R %M115                 (* MEMORI_14 *)
  END_BLK
  MULTIFB
  // as ST:
  //   %TM42(IN := MEMORI_14);
  //   IF %TM42.Q THEN MOVE_Z_2 := FALSE; END_IF;
  //   %TM43(IN := %TM42.Q);
  //   IF %TM43.Q THEN MOVE_X_2 := FALSE; END_IF;
  //   IF %TM43.Q THEN RAISE_6 := TRUE; END_IF;
  //   %TM44(IN := %TM43.Q);
  //   IF %TM44.Q THEN RAISE_6 := FALSE; END_IF;
  //   IF %TM44.Q THEN RIGHT_POS_5 := FALSE; END_IF;
  //   IF %TM44.Q THEN RIGHT_POS_6 := FALSE; END_IF;
  //   IF %TM44.Q THEN MEMORI_14 := FALSE; END_IF;

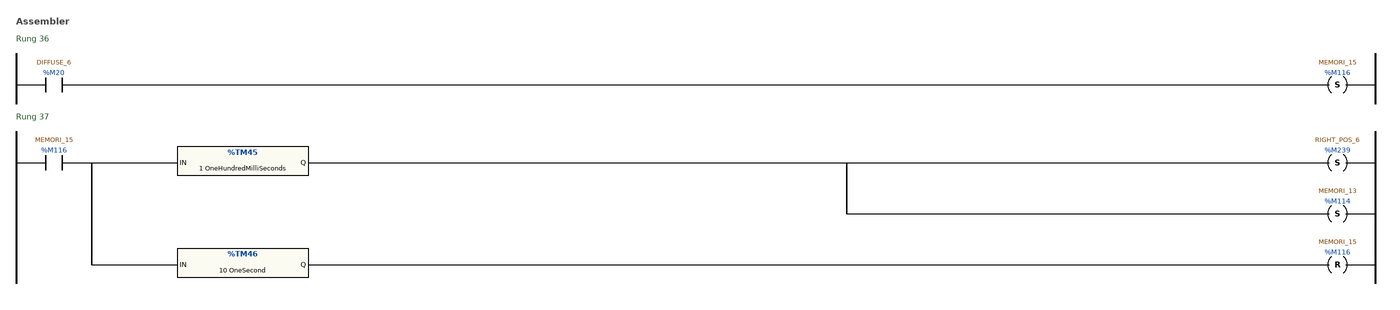

// Rung 36
  LD %M20                 (* DIFFUSE_6 *)
  S %M116                 (* MEMORI_15 *)
  // as ST:
  //   IF DIFFUSE_6 THEN MEMORI_15 := TRUE; END_IF;

// Rung 37
  LD 1
  MULTIFB
  LD 1
  AND %M116               (* MEMORI_15 *)
  ST %MW2009:X0
  BLK %TM45
  LD %MW2009:X0
  IN
  OUT_BLK
  LD Q
  S %M239                 (* RIGHT_POS_6 *)
  S %M114                 (* MEMORI_13 *)
  END_BLK
  BLK %TM46
  LD %MW2009:X0
  IN
  OUT_BLK
  LD Q
  R %M116                 (* MEMORI_15 *)
  END_BLK
  MULTIFB
  // as ST:
  //   %TM45(IN := MEMORI_15);
  //   IF %TM45.Q THEN RIGHT_POS_6 := TRUE; END_IF;
  //   IF %TM45.Q THEN MEMORI_13 := TRUE; END_IF;
  //   %TM46(IN := MEMORI_15);
  //   IF %TM46.Q THEN MEMORI_15 := FALSE; END_IF;

POU Sorting
  (* SectionNumber=3 *)

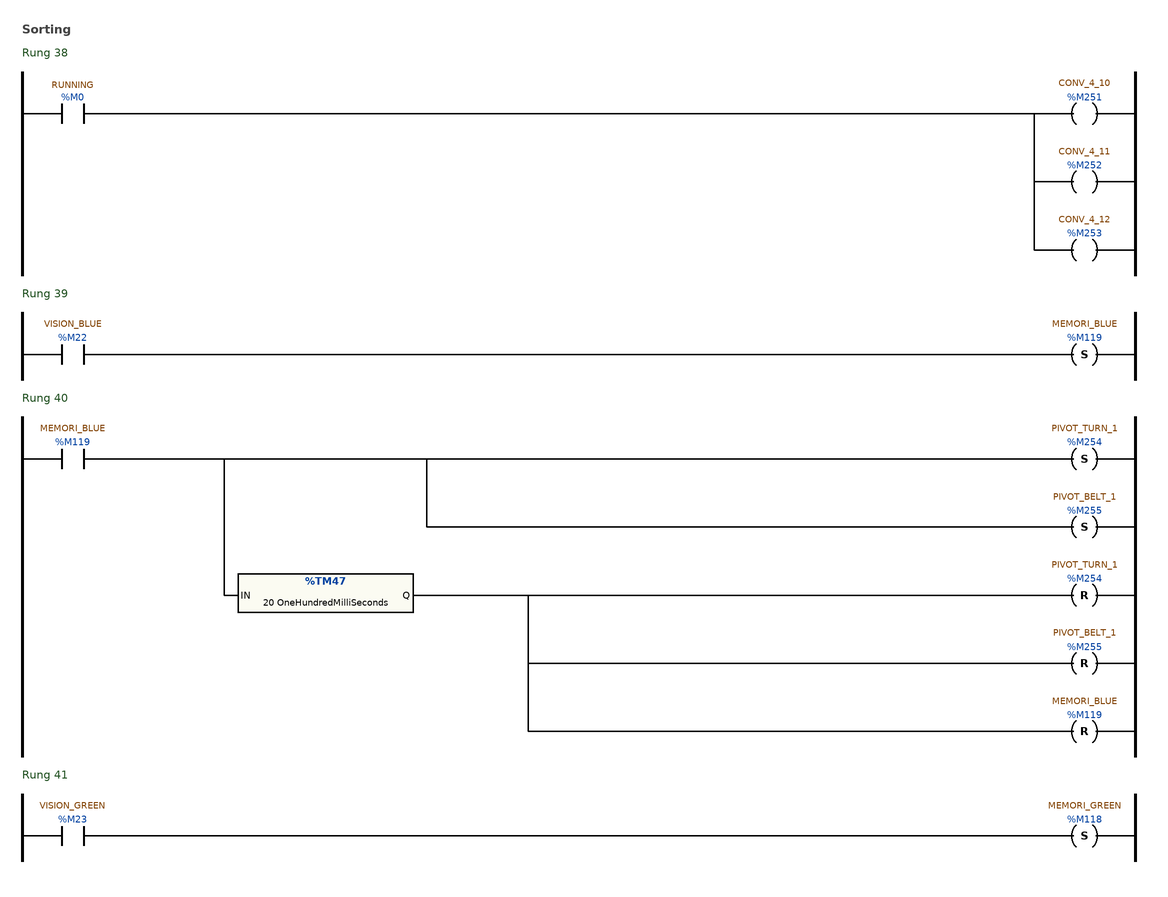

// Rung 38
  LD %M0                  (* RUNNING *)
  ST %M251                (* CONV_4_10 *)
  ST %M252                (* CONV_4_11 *)
  ST %M253                (* CONV_4_12 *)
  // as ST:
  //   CONV_4_10 := RUNNING;
  //   CONV_4_11 := RUNNING;
  //   CONV_4_12 := RUNNING;

// Rung 39
  LD %M22                 (* VISION_BLUE *)
  S %M119                 (* MEMORI_BLUE *)
  // as ST:
  //   IF VISION_BLUE THEN MEMORI_BLUE := TRUE; END_IF;

// Rung 40
  LD 1
  MULTIFB
  LD 1
  AND %M119               (* MEMORI_BLUE *)
  ST %MW2009:X0
  LD %MW2009:X0
  S %M254                 (* PIVOT_TURN_1 *)
  S %M255                 (* PIVOT_BELT_1 *)
  BLK %TM47
  LD %MW2009:X0
  IN
  OUT_BLK
  LD Q
  R %M254                 (* PIVOT_TURN_1 *)
  R %M255                 (* PIVOT_BELT_1 *)
  R %M119                 (* MEMORI_BLUE *)
  END_BLK
  MULTIFB
  // as ST:
  //   IF MEMORI_BLUE THEN PIVOT_TURN_1 := TRUE; END_IF;
  //   IF MEMORI_BLUE THEN PIVOT_BELT_1 := TRUE; END_IF;
  //   %TM47(IN := MEMORI_BLUE);
  //   IF %TM47.Q THEN PIVOT_TURN_1 := FALSE; END_IF;
  //   IF %TM47.Q THEN PIVOT_BELT_1 := FALSE; END_IF;
  //   IF %TM47.Q THEN MEMORI_BLUE := FALSE; END_IF;

// Rung 41
  LD %M23                 (* VISION_GREEN *)
  S %M118                 (* MEMORI_GREEN *)
  // as ST:
  //   IF VISION_GREEN THEN MEMORI_GREEN := TRUE; END_IF;

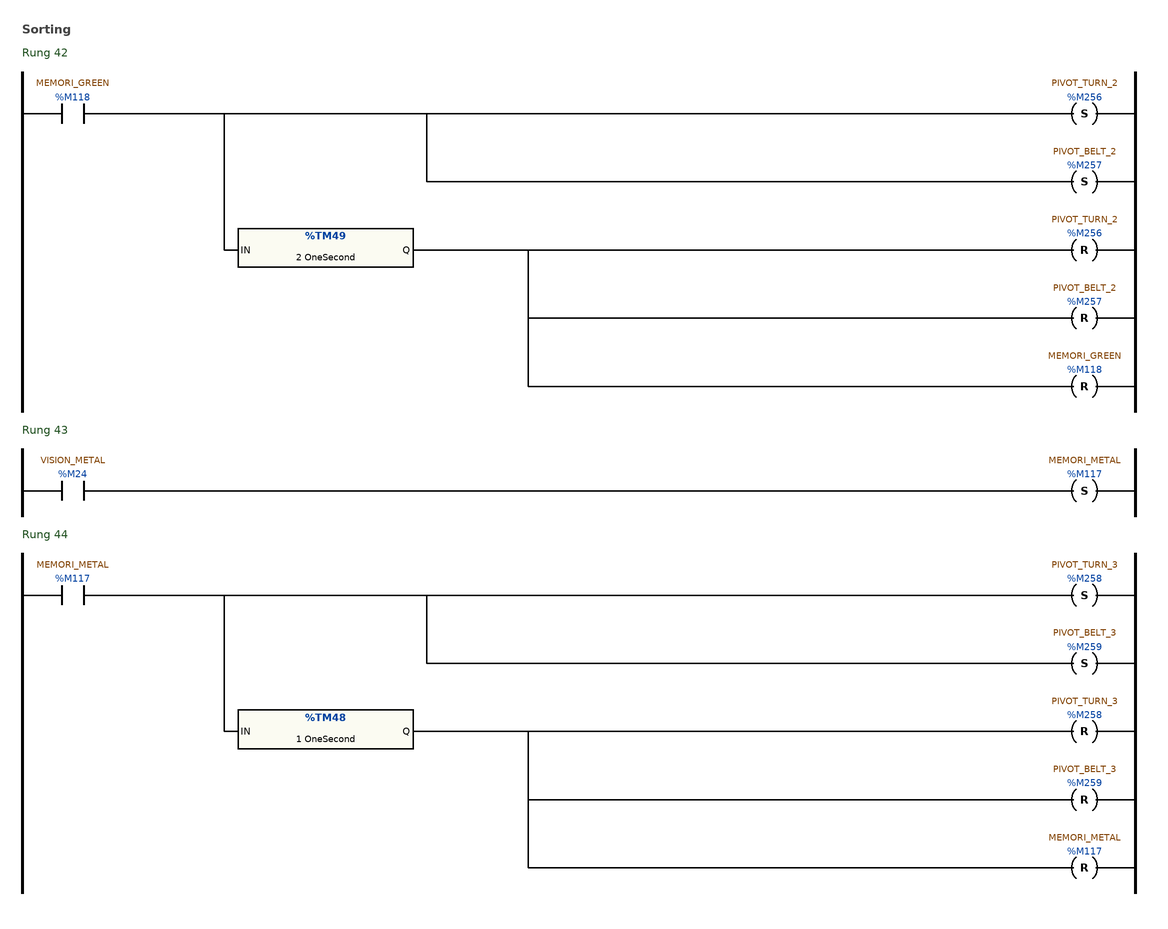

// Rung 42
  LD 1
  MULTIFB
  LD 1
  AND %M118               (* MEMORI_GREEN *)
  ST %MW2009:X0
  LD %MW2009:X0
  S %M256                 (* PIVOT_TURN_2 *)
  S %M257                 (* PIVOT_BELT_2 *)
  BLK %TM49
  LD %MW2009:X0
  IN
  OUT_BLK
  LD Q
  R %M256                 (* PIVOT_TURN_2 *)
  R %M257                 (* PIVOT_BELT_2 *)
  R %M118                 (* MEMORI_GREEN *)
  END_BLK
  MULTIFB
  // as ST:
  //   IF MEMORI_GREEN THEN PIVOT_TURN_2 := TRUE; END_IF;
  //   IF MEMORI_GREEN THEN PIVOT_BELT_2 := TRUE; END_IF;
  //   %TM49(IN := MEMORI_GREEN);
  //   IF %TM49.Q THEN PIVOT_TURN_2 := FALSE; END_IF;
  //   IF %TM49.Q THEN PIVOT_BELT_2 := FALSE; END_IF;
  //   IF %TM49.Q THEN MEMORI_GREEN := FALSE; END_IF;

// Rung 43
  LD %M24                 (* VISION_METAL *)
  S %M117                 (* MEMORI_METAL *)
  // as ST:
  //   IF VISION_METAL THEN MEMORI_METAL := TRUE; END_IF;

// Rung 44
  LD 1
  MULTIFB
  LD 1
  AND %M117               (* MEMORI_METAL *)
  ST %MW2009:X0
  LD %MW2009:X0
  S %M258                 (* PIVOT_TURN_3 *)
  S %M259                 (* PIVOT_BELT_3 *)
  BLK %TM48
  LD %MW2009:X0
  IN
  OUT_BLK
  LD Q
  R %M258                 (* PIVOT_TURN_3 *)
  R %M259                 (* PIVOT_BELT_3 *)
  R %M117                 (* MEMORI_METAL *)
  END_BLK
  MULTIFB
  // as ST:
  //   IF MEMORI_METAL THEN PIVOT_TURN_3 := TRUE; END_IF;
  //   IF MEMORI_METAL THEN PIVOT_BELT_3 := TRUE; END_IF;
  //   %TM48(IN := MEMORI_METAL);
  //   IF %TM48.Q THEN PIVOT_TURN_3 := FALSE; END_IF;
  //   IF %TM48.Q THEN PIVOT_BELT_3 := FALSE; END_IF;
  //   IF %TM48.Q THEN MEMORI_METAL := FALSE; END_IF;
